PROGRAM P_Inputs
VAR
	fbJoystickLeftVert 					: FB_JoystickInputScaling;
	fbJoystickLeftHor 					: FB_JoystickInputScaling;
	
	fbJoystickRightVert 				: FB_JoystickInputScaling;
	fbJoystickRightHor 					: FB_JoystickInputScaling;
	
	
END_VAR

 fbJoystickLeftVert(
	bEnable := G_Work.bManualMode,
	nRawInput := G_Inputs.stJoyLY.nValue,
	stJoystickInputScaling := G_Parameters.stParam.stJoystickInputScalingLeftY,
	fNormalizedOutput => G_Sensors.fJoystickLeftNormalizedY
);

fbJoystickLeftHor(
	bEnable := G_Work.bManualMode,
	nRawInput := G_Inputs.stJoyLX.nValue,
	stJoystickInputScaling := G_Parameters.stParam.stJoystickInputScalingLeftX,
	fNormalizedOutput => G_Sensors.fJoystickLeftNormalizedX
);

IF G_Sensors.fJoystickLeftNormalizedX < 0 THEN
	G_Sensors.MCDirectionAxis1 := MC_Positive_Direction;
ELSIF G_Sensors.fJoystickLeftNormalizedX > 0 THEN
	G_Sensors.MCDirectionAxis1 := MC_Negative_Direction;	
//ELSE
//	G_Sensors.MCDirectionAxis1 := MC_Current_Direction;
END_IF


fbJoystickRightVert(
	bEnable := G_Work.bManualMode,
	nRawInput := G_Inputs.stJoyRY.nValue,
	stJoystickInputScaling := G_Parameters.stParam.stJoystickInputScalingRightY,
	fNormalizedOutput => G_Sensors.fJoystickRightNormalizedY
);

fbJoystickRightHor(
	bEnable := G_Work.bManualMode,
	nRawInput := G_Inputs.stJoyRX.nValue,
	stJoystickInputScaling := G_Parameters.stParam.stJoystickInputScalingRightX,
	fNormalizedOutput => G_Sensors.fJoystickRightNormalizedX
);

END_PROGRAM

(* stored: Version 1.1.0.1, ProductVersion 3.1.4024.12
   POU P_Inputs: Id {8b676dbd-393f-42d6-8803-330b6e90ab14}, SpecialFunc None *)
